// TIA Portal V21 export
FUNCTION "OUTPUT" : Void   // FC4, LAD
{ S7_Optimized_Access := 'TRUE' }
// stored: SetENOAutomatically false
   VAR_TEMP   // added for the SCL form of the ladder/FBD networks
      _w1 : Bool;
   END_VAR
BEGIN

REGION Network 1: VCC PUMP
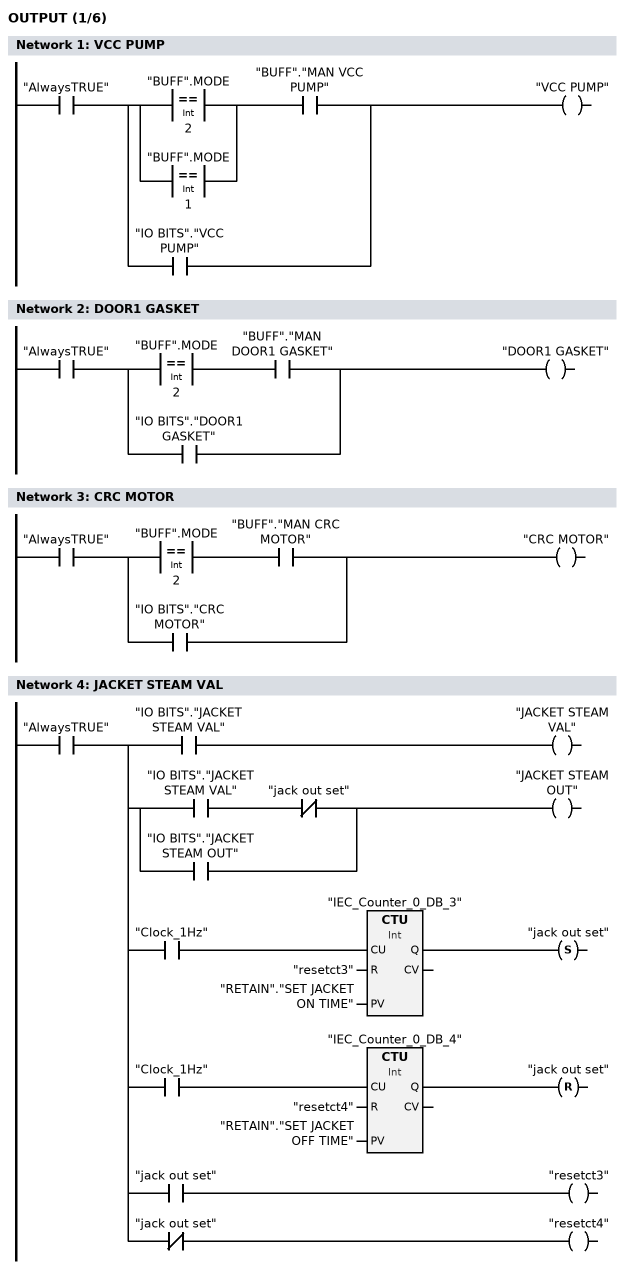
   RUNG wire#powerrail
      Contact( "AlwaysTRUE" )
      wire#w1
      { S7_Templates := "SrcType := Int" } EQ_Contact(in1 := "BUFF".MODE, in2 := 2)
      wire#w2
      Contact( "BUFF"."MAN VCC PUMP" )
      wire#w3
      Coil( "VCC PUMP" )
   END_RUNG
   RUNG wire#w1
      { S7_Templates := "SrcType := Int" } EQ_Contact(in1 := "BUFF".MODE, in2 := 1)
   END_RUNG wire#w2
   RUNG wire#w1
      Contact( "IO BITS"."VCC PUMP" )
   END_RUNG wire#w3
   // the same network as SCL:
   "VCC PUMP" := "AlwaysTRUE" AND (((("BUFF".MODE = 2) OR ("BUFF".MODE = 1)) AND "BUFF"."MAN VCC PUMP") OR "IO BITS"."VCC PUMP");
END_REGION

REGION Network 2: DOOR1 GASKET
   RUNG wire#powerrail
      Contact( "AlwaysTRUE" )
      wire#w1
      { S7_Templates := "SrcType := Int" } EQ_Contact(in1 := "BUFF".MODE, in2 := 2)
      Contact( "BUFF"."MAN DOOR1 GASKET" )
      wire#w2
      Coil( "DOOR1 GASKET" )
   END_RUNG
   RUNG wire#w1
      Contact( "IO BITS"."DOOR1 GASKET" )
   END_RUNG wire#w2
   // the same network as SCL:
   "DOOR1 GASKET" := "AlwaysTRUE" AND ((("BUFF".MODE = 2) AND "BUFF"."MAN DOOR1 GASKET") OR "IO BITS"."DOOR1 GASKET");
END_REGION

REGION Network 3: CRC MOTOR
   RUNG wire#powerrail
      Contact( "AlwaysTRUE" )
      wire#w1
      { S7_Templates := "SrcType := Int" } EQ_Contact(in1 := "BUFF".MODE, in2 := 2)
      Contact( "BUFF"."MAN CRC MOTOR" )
      wire#w2
      Coil( "CRC MOTOR" )
   END_RUNG
   RUNG wire#w1
      Contact( "IO BITS"."CRC MOTOR" )
   END_RUNG wire#w2
   // the same network as SCL:
   "CRC MOTOR" := "AlwaysTRUE" AND ((("BUFF".MODE = 2) AND "BUFF"."MAN CRC MOTOR") OR "IO BITS"."CRC MOTOR");
END_REGION

REGION Network 4: JACKET STEAM VAL
   RUNG wire#powerrail
      Contact( "AlwaysTRUE" )
      wire#w1
      Contact( "IO BITS"."JACKET STEAM VAL" )
      Coil( "JACKET STEAM VAL" )
   END_RUNG
   RUNG wire#w1
      Contact( "IO BITS"."JACKET STEAM VAL" )
      I_Contact( "jack out set" )
      wire#w2
      Coil( "JACKET STEAM OUT" )
   END_RUNG
   RUNG wire#w1
      Contact( "IO BITS"."JACKET STEAM OUT" )
   END_RUNG wire#w2
   RUNG wire#w1
      Contact( "Clock_1Hz" )
      { S7_Templates := "value_type := Int" } "IEC_Counter_0_DB_3".CTU(r := "resetct3", pv := "RETAIN"."SET JACKET ON TIME", cv =>)
      S_Coil( "jack out set" )
   END_RUNG
   RUNG wire#w1
      Contact( "Clock_1Hz" )
      { S7_Templates := "value_type := Int" } "IEC_Counter_0_DB_4".CTU(r := "resetct4", pv := "RETAIN"."SET JACKET OFF TIME", cv =>)
      R_Coil( "jack out set" )
   END_RUNG
   RUNG wire#w1
      Contact( "jack out set" )
      Coil( "resetct3" )
   END_RUNG
   RUNG wire#w1
      I_Contact( "jack out set" )
      Coil( "resetct4" )
   END_RUNG
   // the same network as SCL:
   "JACKET STEAM VAL" := "AlwaysTRUE" AND "IO BITS"."JACKET STEAM VAL";
   "JACKET STEAM OUT" := "AlwaysTRUE" AND (("IO BITS"."JACKET STEAM VAL" AND NOT "jack out set") OR "IO BITS"."JACKET STEAM OUT");
   "IEC_Counter_0_DB_3".CTU(CU := "AlwaysTRUE" AND "Clock_1Hz",
                           R := "resetct3",
                           PV := "RETAIN"."SET JACKET ON TIME");
   IF "IEC_Counter_0_DB_3".Q THEN "jack out set" := TRUE; END_IF;
   "IEC_Counter_0_DB_4".CTU(CU := "AlwaysTRUE" AND "Clock_1Hz",
                           R := "resetct4",
                           PV := "RETAIN"."SET JACKET OFF TIME");
   IF "IEC_Counter_0_DB_4".Q THEN "jack out set" := FALSE; END_IF;
   "resetct3" := "AlwaysTRUE" AND "jack out set";
   "resetct4" := "AlwaysTRUE" AND NOT "jack out set";
END_REGION

REGION Network 5: CHAMBER STEAM VAL
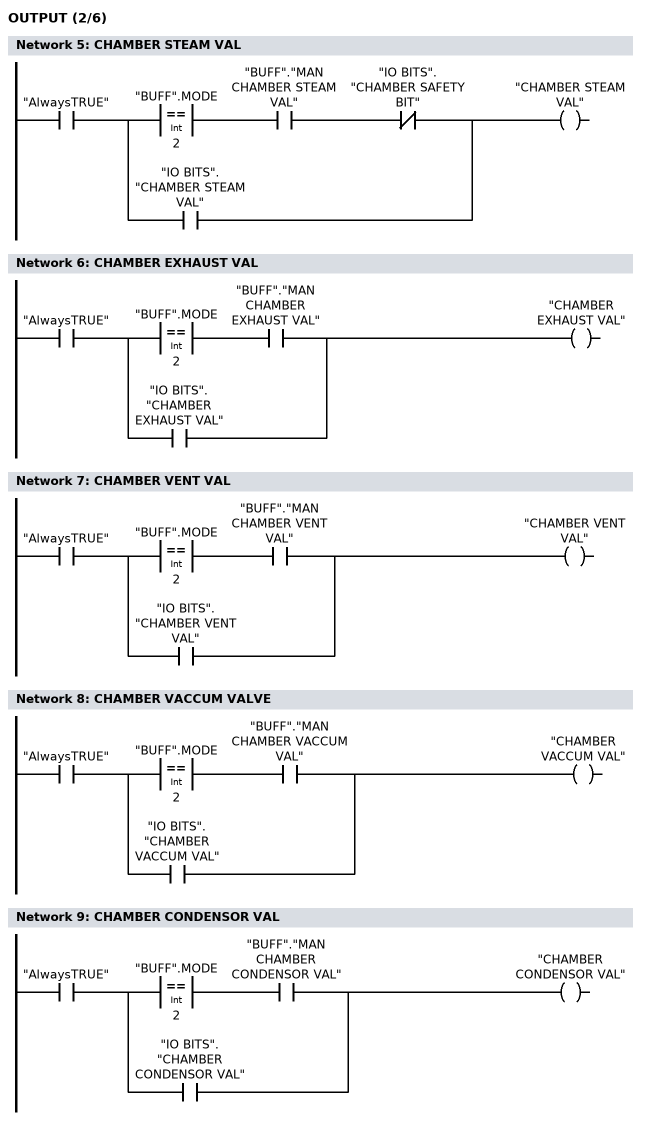
   RUNG wire#powerrail
      Contact( "AlwaysTRUE" )
      wire#w1
      { S7_Templates := "SrcType := Int" } EQ_Contact(in1 := "BUFF".MODE, in2 := 2)
      Contact( "BUFF"."MAN CHAMBER STEAM VAL" )
      I_Contact( "IO BITS"."CHAMBER SAFETY BIT" )
      wire#w2
      Coil( "CHAMBER STEAM VAL" )
   END_RUNG
   RUNG wire#w1
      Contact( "IO BITS"."CHAMBER STEAM VAL" )
   END_RUNG wire#w2
   // the same network as SCL:
   "CHAMBER STEAM VAL" := "AlwaysTRUE" AND ((("BUFF".MODE = 2) AND "BUFF"."MAN CHAMBER STEAM VAL" AND NOT "IO BITS"."CHAMBER SAFETY BIT") OR "IO BITS"."CHAMBER STEAM VAL");
END_REGION

REGION Network 6: CHAMBER EXHAUST VAL
   RUNG wire#powerrail
      Contact( "AlwaysTRUE" )
      wire#w1
      { S7_Templates := "SrcType := Int" } EQ_Contact(in1 := "BUFF".MODE, in2 := 2)
      Contact( "BUFF"."MAN CHAMBER EXHAUST VAL" )
      wire#w2
      Coil( "CHAMBER EXHAUST VAL" )
   END_RUNG
   RUNG wire#w1
      Contact( "IO BITS"."CHAMBER EXHAUST VAL" )
   END_RUNG wire#w2
   // the same network as SCL:
   "CHAMBER EXHAUST VAL" := "AlwaysTRUE" AND ((("BUFF".MODE = 2) AND "BUFF"."MAN CHAMBER EXHAUST VAL") OR "IO BITS"."CHAMBER EXHAUST VAL");
END_REGION

REGION Network 7: CHAMBER VENT VAL
   RUNG wire#powerrail
      Contact( "AlwaysTRUE" )
      wire#w1
      { S7_Templates := "SrcType := Int" } EQ_Contact(in1 := "BUFF".MODE, in2 := 2)
      Contact( "BUFF"."MAN CHAMBER VENT VAL" )
      wire#w2
      Coil( "CHAMBER VENT VAL" )
   END_RUNG
   RUNG wire#w1
      Contact( "IO BITS"."CHAMBER VENT VAL" )
   END_RUNG wire#w2
   // the same network as SCL:
   "CHAMBER VENT VAL" := "AlwaysTRUE" AND ((("BUFF".MODE = 2) AND "BUFF"."MAN CHAMBER VENT VAL") OR "IO BITS"."CHAMBER VENT VAL");
END_REGION

REGION Network 8: CHAMBER VACCUM VALVE
   RUNG wire#powerrail
      Contact( "AlwaysTRUE" )
      wire#w1
      { S7_Templates := "SrcType := Int" } EQ_Contact(in1 := "BUFF".MODE, in2 := 2)
      Contact( "BUFF"."MAN CHAMBER VACCUM VAL" )
      wire#w2
      Coil( "CHAMBER VACCUM VAL" )
   END_RUNG
   RUNG wire#w1
      Contact( "IO BITS"."CHAMBER VACCUM VAL" )
   END_RUNG wire#w2
   // the same network as SCL:
   "CHAMBER VACCUM VAL" := "AlwaysTRUE" AND ((("BUFF".MODE = 2) AND "BUFF"."MAN CHAMBER VACCUM VAL") OR "IO BITS"."CHAMBER VACCUM VAL");
END_REGION

REGION Network 9: CHAMBER CONDENSOR VAL
   RUNG wire#powerrail
      Contact( "AlwaysTRUE" )
      wire#w1
      { S7_Templates := "SrcType := Int" } EQ_Contact(in1 := "BUFF".MODE, in2 := 2)
      Contact( "BUFF"."MAN CHAMBER CONDENSOR VAL" )
      wire#w2
      Coil( "CHAMBER CONDENSOR VAL" )
   END_RUNG
   RUNG wire#w1
      Contact( "IO BITS"."CHAMBER CONDENSOR VAL" )
   END_RUNG wire#w2
   // the same network as SCL:
   "CHAMBER CONDENSOR VAL" := "AlwaysTRUE" AND ((("BUFF".MODE = 2) AND "BUFF"."MAN CHAMBER CONDENSOR VAL") OR "IO BITS"."CHAMBER CONDENSOR VAL");
END_REGION

REGION Network 10: process on lamp
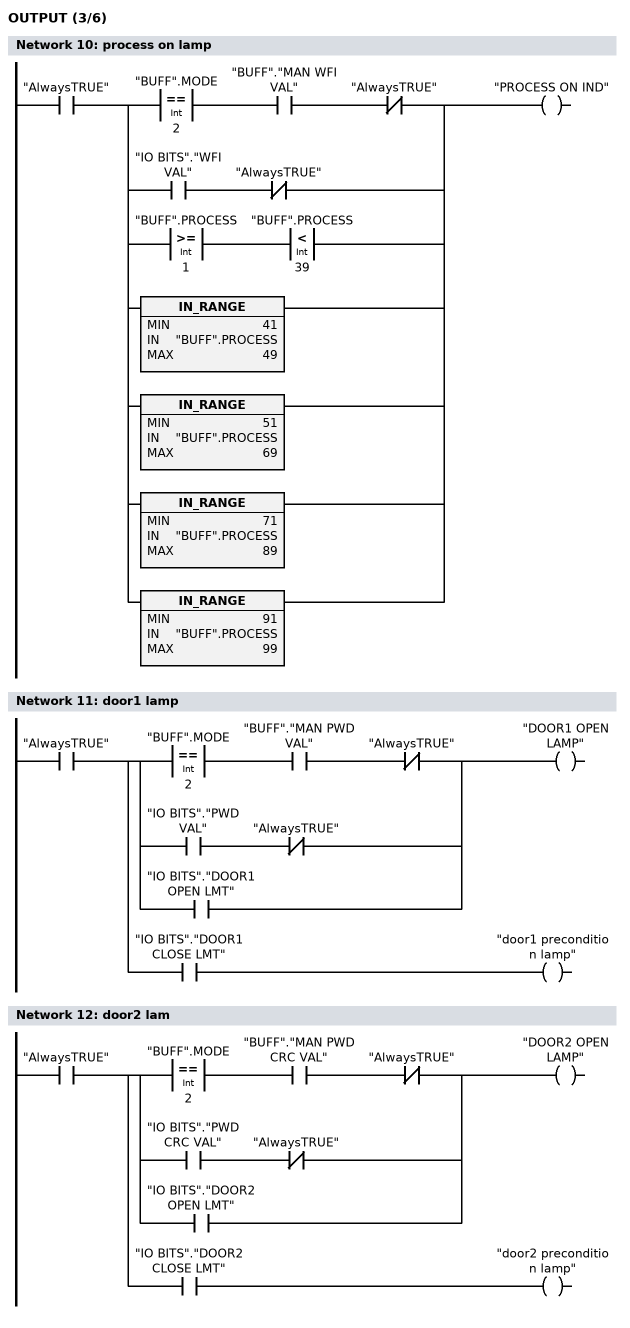
   RUNG wire#powerrail
      Contact( "AlwaysTRUE" )
      wire#w1
      { S7_Templates := "SrcType := Int" } EQ_Contact(in1 := "BUFF".MODE, in2 := 2)
      Contact( "BUFF"."MAN WFI VAL" )
      I_Contact( "AlwaysTRUE" )
      wire#w2
      Coil( "PROCESS ON IND" )
   END_RUNG
   RUNG wire#w1
      Contact( "IO BITS"."WFI VAL" )
      I_Contact( "AlwaysTRUE" )
   END_RUNG wire#w2
   RUNG wire#w1
      { S7_Templates := "SrcType := Int" } GE_Contact(in1 := "BUFF".PROCESS, in2 := 1)
      { S7_Templates := "SrcType := Int" } LT_Contact(in1 := "BUFF".PROCESS, in2 := 39)
   END_RUNG wire#w2
   RUNG wire#w1
      { S7_Templates := "SrcType := Int" } InRange(min := 41, in := "BUFF".PROCESS, max := 49)
   END_RUNG wire#w2
   RUNG wire#w1
      { S7_Templates := "SrcType := Int" } InRange(min := 51, in := "BUFF".PROCESS, max := 69)
   END_RUNG wire#w2
   RUNG wire#w1
      { S7_Templates := "SrcType := Int" } InRange(min := 71, in := "BUFF".PROCESS, max := 89)
   END_RUNG wire#w2
   RUNG wire#w1
      { S7_Templates := "SrcType := Int" } InRange(min := 91, in := "BUFF".PROCESS, max := 99)
   END_RUNG wire#w2
   // the same network as SCL:
   "PROCESS ON IND" := "AlwaysTRUE" AND ((("BUFF".MODE = 2) AND "BUFF"."MAN WFI VAL" AND NOT "AlwaysTRUE") OR ("IO BITS"."WFI VAL" AND NOT "AlwaysTRUE") OR (("BUFF".PROCESS >= 1) AND ("BUFF".PROCESS < 39)) OR ((41 <= "BUFF".PROCESS) AND ("BUFF".PROCESS <= 49)) OR ((51 <= "BUFF".PROCESS) AND ("BUFF".PROCESS <= 69)) OR ((71 <= "BUFF".PROCESS) AND ("BUFF".PROCESS <= 89)) OR ((91 <= "BUFF".PROCESS) AND ("BUFF".PROCESS <= 99)));
END_REGION

REGION Network 11: door1 lamp
   RUNG wire#powerrail
      Contact( "AlwaysTRUE" )
      wire#w1
      { S7_Templates := "SrcType := Int" } EQ_Contact(in1 := "BUFF".MODE, in2 := 2)
      Contact( "BUFF"."MAN PWD VAL" )
      I_Contact( "AlwaysTRUE" )
      wire#w2
      Coil( "DOOR1 OPEN LAMP" )
   END_RUNG
   RUNG wire#w1
      Contact( "IO BITS"."PWD VAL" )
      I_Contact( "AlwaysTRUE" )
   END_RUNG wire#w2
   RUNG wire#w1
      Contact( "IO BITS"."DOOR1 OPEN LMT" )
   END_RUNG wire#w2
   RUNG wire#w1
      Contact( "IO BITS"."DOOR1 CLOSE LMT" )
      Coil( "door1 precondition lamp" )
   END_RUNG
   // the same network as SCL:
   "DOOR1 OPEN LAMP" := "AlwaysTRUE" AND ((("BUFF".MODE = 2) AND "BUFF"."MAN PWD VAL" AND NOT "AlwaysTRUE") OR ("IO BITS"."PWD VAL" AND NOT "AlwaysTRUE") OR "IO BITS"."DOOR1 OPEN LMT");
   "door1 precondition lamp" := "AlwaysTRUE" AND "IO BITS"."DOOR1 CLOSE LMT";
END_REGION

REGION Network 12: door2 lam
   RUNG wire#powerrail
      Contact( "AlwaysTRUE" )
      wire#w1
      { S7_Templates := "SrcType := Int" } EQ_Contact(in1 := "BUFF".MODE, in2 := 2)
      Contact( "BUFF"."MAN PWD CRC VAL" )
      I_Contact( "AlwaysTRUE" )
      wire#w2
      Coil( "DOOR2 OPEN LAMP" )
   END_RUNG
   RUNG wire#w1
      Contact( "IO BITS"."PWD CRC VAL" )
      I_Contact( "AlwaysTRUE" )
   END_RUNG wire#w2
   RUNG wire#w1
      Contact( "IO BITS"."DOOR2 OPEN LMT" )
   END_RUNG wire#w2
   RUNG wire#w1
      Contact( "IO BITS"."DOOR2 CLOSE LMT" )
      Coil( "door2 precondition lamp" )
   END_RUNG
   // the same network as SCL:
   "DOOR2 OPEN LAMP" := "AlwaysTRUE" AND ((("BUFF".MODE = 2) AND "BUFF"."MAN PWD CRC VAL" AND NOT "AlwaysTRUE") OR ("IO BITS"."PWD CRC VAL" AND NOT "AlwaysTRUE") OR "IO BITS"."DOOR2 OPEN LMT");
   "door2 precondition lamp" := "AlwaysTRUE" AND "IO BITS"."DOOR2 CLOSE LMT";
END_REGION

REGION Network 13: DETERGENT DSG VAL
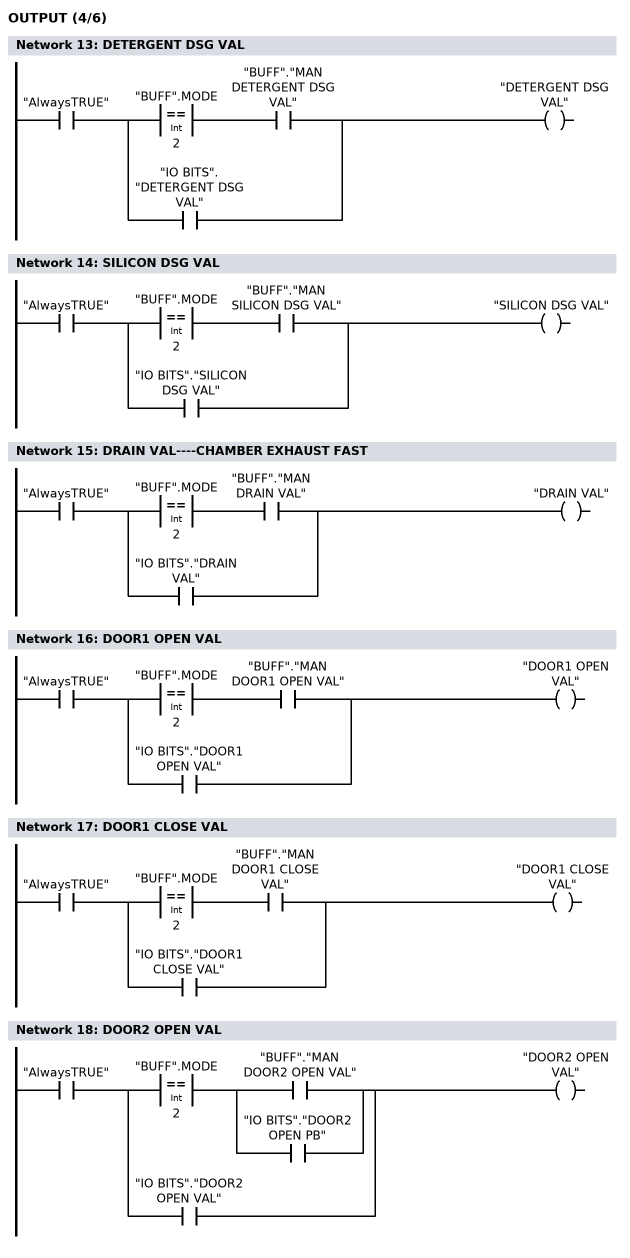
   RUNG wire#powerrail
      Contact( "AlwaysTRUE" )
      wire#w1
      { S7_Templates := "SrcType := Int" } EQ_Contact(in1 := "BUFF".MODE, in2 := 2)
      Contact( "BUFF"."MAN DETERGENT DSG VAL" )
      wire#w2
      Coil( "DETERGENT DSG VAL" )
   END_RUNG
   RUNG wire#w1
      Contact( "IO BITS"."DETERGENT DSG VAL" )
   END_RUNG wire#w2
   // the same network as SCL:
   "DETERGENT DSG VAL" := "AlwaysTRUE" AND ((("BUFF".MODE = 2) AND "BUFF"."MAN DETERGENT DSG VAL") OR "IO BITS"."DETERGENT DSG VAL");
END_REGION

REGION Network 14: SILICON DSG VAL
   RUNG wire#powerrail
      Contact( "AlwaysTRUE" )
      wire#w1
      { S7_Templates := "SrcType := Int" } EQ_Contact(in1 := "BUFF".MODE, in2 := 2)
      Contact( "BUFF"."MAN SILICON DSG VAL" )
      wire#w2
      Coil( "SILICON DSG VAL" )
   END_RUNG
   RUNG wire#w1
      Contact( "IO BITS"."SILICON DSG VAL" )
   END_RUNG wire#w2
   // the same network as SCL:
   "SILICON DSG VAL" := "AlwaysTRUE" AND ((("BUFF".MODE = 2) AND "BUFF"."MAN SILICON DSG VAL") OR "IO BITS"."SILICON DSG VAL");
END_REGION

REGION Network 15: DRAIN VAL----CHAMBER EXHAUST FAST
   RUNG wire#powerrail
      Contact( "AlwaysTRUE" )
      wire#w1
      { S7_Templates := "SrcType := Int" } EQ_Contact(in1 := "BUFF".MODE, in2 := 2)
      Contact( "BUFF"."MAN DRAIN VAL" )
      wire#w2
      Coil( "DRAIN VAL" )
   END_RUNG
   RUNG wire#w1
      Contact( "IO BITS"."DRAIN VAL" )
   END_RUNG wire#w2
   // the same network as SCL:
   "DRAIN VAL" := "AlwaysTRUE" AND ((("BUFF".MODE = 2) AND "BUFF"."MAN DRAIN VAL") OR "IO BITS"."DRAIN VAL");
END_REGION

REGION Network 16: DOOR1 OPEN VAL
   RUNG wire#powerrail
      Contact( "AlwaysTRUE" )
      wire#w1
      { S7_Templates := "SrcType := Int" } EQ_Contact(in1 := "BUFF".MODE, in2 := 2)
      Contact( "BUFF"."MAN DOOR1 OPEN VAL" )
      wire#w2
      Coil( "DOOR1 OPEN VAL" )
   END_RUNG
   RUNG wire#w1
      Contact( "IO BITS"."DOOR1 OPEN VAL" )
   END_RUNG wire#w2
   // the same network as SCL:
   "DOOR1 OPEN VAL" := "AlwaysTRUE" AND ((("BUFF".MODE = 2) AND "BUFF"."MAN DOOR1 OPEN VAL") OR "IO BITS"."DOOR1 OPEN VAL");
END_REGION

REGION Network 17: DOOR1 CLOSE VAL
   RUNG wire#powerrail
      Contact( "AlwaysTRUE" )
      wire#w1
      { S7_Templates := "SrcType := Int" } EQ_Contact(in1 := "BUFF".MODE, in2 := 2)
      Contact( "BUFF"."MAN DOOR1 CLOSE VAL" )
      wire#w2
      Coil( "DOOR1 CLOSE VAL" )
   END_RUNG
   RUNG wire#w1
      Contact( "IO BITS"."DOOR1 CLOSE VAL" )
   END_RUNG wire#w2
   // the same network as SCL:
   "DOOR1 CLOSE VAL" := "AlwaysTRUE" AND ((("BUFF".MODE = 2) AND "BUFF"."MAN DOOR1 CLOSE VAL") OR "IO BITS"."DOOR1 CLOSE VAL");
END_REGION

REGION Network 18: DOOR2 OPEN VAL
   RUNG wire#powerrail
      Contact( "AlwaysTRUE" )
      wire#w1
      { S7_Templates := "SrcType := Int" } EQ_Contact(in1 := "BUFF".MODE, in2 := 2)
      wire#w2
      Contact( "BUFF"."MAN DOOR2 OPEN VAL" )
      wire#w3
      Coil( "DOOR2 OPEN VAL" )
   END_RUNG
   RUNG wire#w2
      Contact( "IO BITS"."DOOR2 OPEN PB" )
   END_RUNG wire#w3
   RUNG wire#w1
      Contact( "IO BITS"."DOOR2 OPEN VAL" )
   END_RUNG wire#w3
   // the same network as SCL:
   "DOOR2 OPEN VAL" := "AlwaysTRUE" AND ((("BUFF".MODE = 2) AND ("BUFF"."MAN DOOR2 OPEN VAL" OR "IO BITS"."DOOR2 OPEN PB")) OR "IO BITS"."DOOR2 OPEN VAL");
END_REGION

REGION Network 19: DOOR2 CLOSE VAL
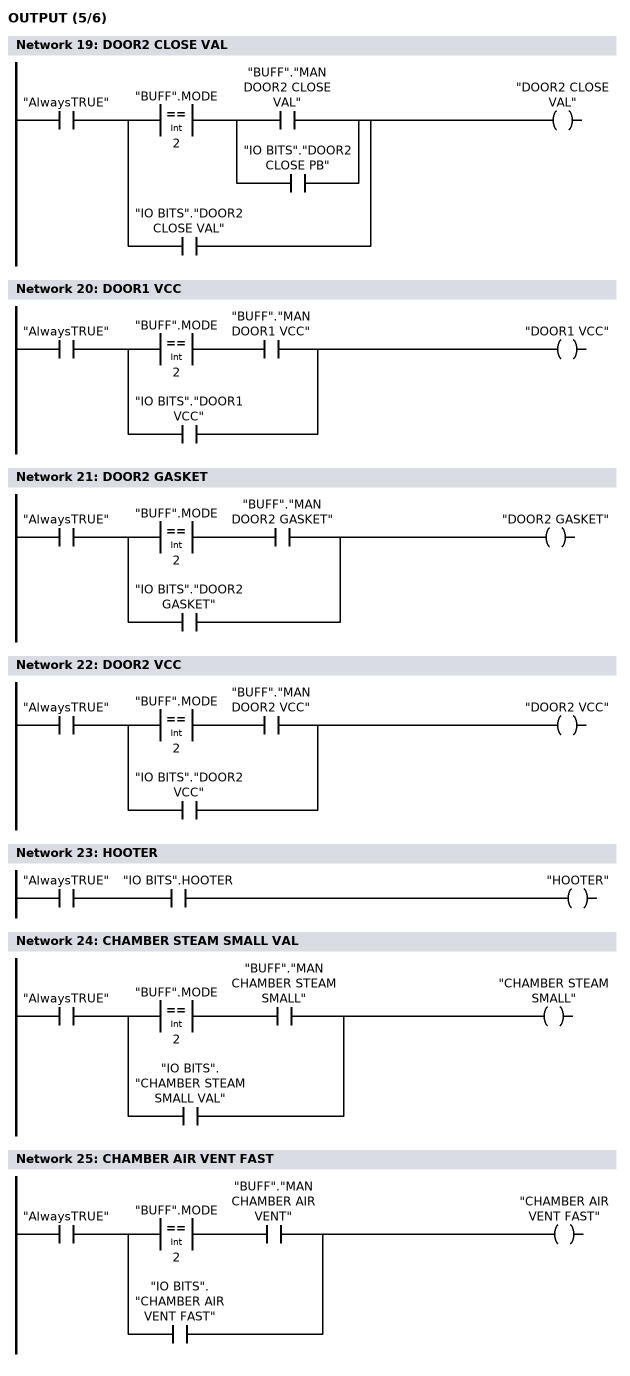
   RUNG wire#powerrail
      Contact( "AlwaysTRUE" )
      wire#w1
      { S7_Templates := "SrcType := Int" } EQ_Contact(in1 := "BUFF".MODE, in2 := 2)
      wire#w2
      Contact( "BUFF"."MAN DOOR2 CLOSE VAL" )
      wire#w3
      Coil( "DOOR2 CLOSE VAL" )
   END_RUNG
   RUNG wire#w2
      Contact( "IO BITS"."DOOR2 CLOSE PB" )
   END_RUNG wire#w3
   RUNG wire#w1
      Contact( "IO BITS"."DOOR2 CLOSE VAL" )
   END_RUNG wire#w3
   // the same network as SCL:
   "DOOR2 CLOSE VAL" := "AlwaysTRUE" AND ((("BUFF".MODE = 2) AND ("BUFF"."MAN DOOR2 CLOSE VAL" OR "IO BITS"."DOOR2 CLOSE PB")) OR "IO BITS"."DOOR2 CLOSE VAL");
END_REGION

REGION Network 20: DOOR1 VCC
   RUNG wire#powerrail
      Contact( "AlwaysTRUE" )
      wire#w1
      { S7_Templates := "SrcType := Int" } EQ_Contact(in1 := "BUFF".MODE, in2 := 2)
      Contact( "BUFF"."MAN DOOR1 VCC" )
      wire#w2
      Coil( "DOOR1 VCC" )
   END_RUNG
   RUNG wire#w1
      Contact( "IO BITS"."DOOR1 VCC" )
   END_RUNG wire#w2
   // the same network as SCL:
   "DOOR1 VCC" := "AlwaysTRUE" AND ((("BUFF".MODE = 2) AND "BUFF"."MAN DOOR1 VCC") OR "IO BITS"."DOOR1 VCC");
END_REGION

REGION Network 21: DOOR2 GASKET
   RUNG wire#powerrail
      Contact( "AlwaysTRUE" )
      wire#w1
      { S7_Templates := "SrcType := Int" } EQ_Contact(in1 := "BUFF".MODE, in2 := 2)
      Contact( "BUFF"."MAN DOOR2 GASKET" )
      wire#w2
      Coil( "DOOR2 GASKET" )
   END_RUNG
   RUNG wire#w1
      Contact( "IO BITS"."DOOR2 GASKET" )
   END_RUNG wire#w2
   // the same network as SCL:
   "DOOR2 GASKET" := "AlwaysTRUE" AND ((("BUFF".MODE = 2) AND "BUFF"."MAN DOOR2 GASKET") OR "IO BITS"."DOOR2 GASKET");
END_REGION

REGION Network 22: DOOR2 VCC
   RUNG wire#powerrail
      Contact( "AlwaysTRUE" )
      wire#w1
      { S7_Templates := "SrcType := Int" } EQ_Contact(in1 := "BUFF".MODE, in2 := 2)
      Contact( "BUFF"."MAN DOOR2 VCC" )
      wire#w2
      Coil( "DOOR2 VCC" )
   END_RUNG
   RUNG wire#w1
      Contact( "IO BITS"."DOOR2 VCC" )
   END_RUNG wire#w2
   // the same network as SCL:
   "DOOR2 VCC" := "AlwaysTRUE" AND ((("BUFF".MODE = 2) AND "BUFF"."MAN DOOR2 VCC") OR "IO BITS"."DOOR2 VCC");
END_REGION

REGION Network 23: HOOTER
   RUNG wire#powerrail
      Contact( "AlwaysTRUE" )
      Contact( "IO BITS".HOOTER )
      Coil( "HOOTER" )
   END_RUNG
   // the same network as SCL:
   "HOOTER" := "AlwaysTRUE" AND "IO BITS".HOOTER;
END_REGION

REGION Network 24: CHAMBER STEAM SMALL VAL
   RUNG wire#powerrail
      Contact( "AlwaysTRUE" )
      wire#w1
      { S7_Templates := "SrcType := Int" } EQ_Contact(in1 := "BUFF".MODE, in2 := 2)
      Contact( "BUFF"."MAN CHAMBER STEAM SMALL" )
      wire#w2
      Coil( "CHAMBER STEAM SMALL" )
   END_RUNG
   RUNG wire#w1
      Contact( "IO BITS"."CHAMBER STEAM SMALL VAL" )
   END_RUNG wire#w2
   // the same network as SCL:
   "CHAMBER STEAM SMALL" := "AlwaysTRUE" AND ((("BUFF".MODE = 2) AND "BUFF"."MAN CHAMBER STEAM SMALL") OR "IO BITS"."CHAMBER STEAM SMALL VAL");
END_REGION

REGION Network 25: CHAMBER AIR VENT FAST
   RUNG wire#powerrail
      Contact( "AlwaysTRUE" )
      wire#w1
      { S7_Templates := "SrcType := Int" } EQ_Contact(in1 := "BUFF".MODE, in2 := 2)
      Contact( "BUFF"."MAN CHAMBER AIR VENT" )
      wire#w2
      Coil( "CHAMBER AIR VENT FAST" )
   END_RUNG
   RUNG wire#w1
      Contact( "IO BITS"."CHAMBER AIR VENT FAST" )
   END_RUNG wire#w2
   // the same network as SCL:
   "CHAMBER AIR VENT FAST" := "AlwaysTRUE" AND ((("BUFF".MODE = 2) AND "BUFF"."MAN CHAMBER AIR VENT") OR "IO BITS"."CHAMBER AIR VENT FAST");
END_REGION

REGION Network 26: BOILER
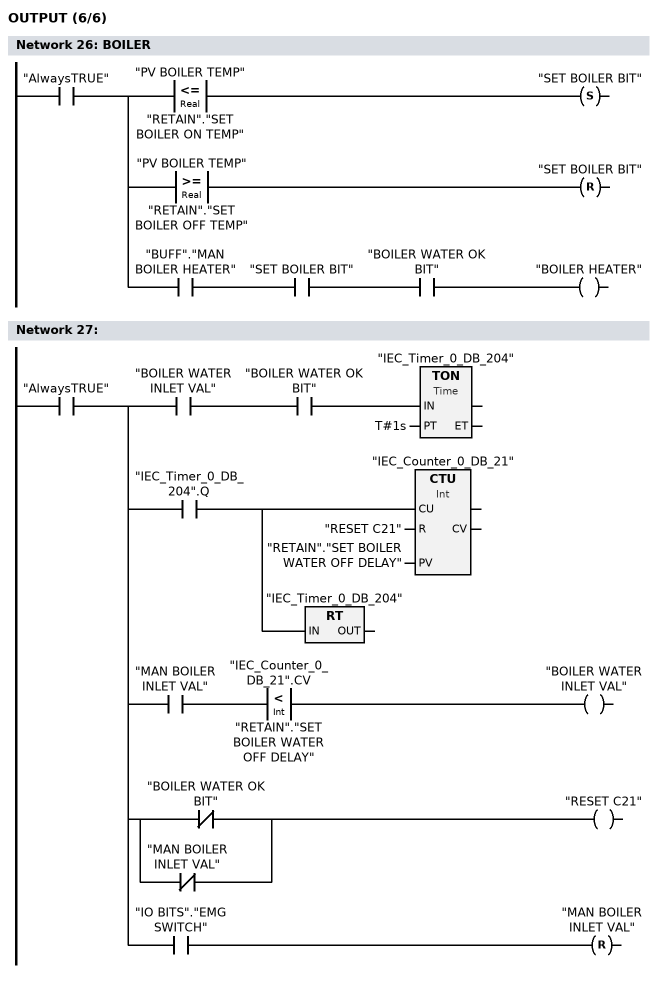
   RUNG wire#powerrail
      Contact( "AlwaysTRUE" )
      wire#w1
      { S7_Templates := "SrcType := Real" } LE_Contact(in1 := "PV BOILER TEMP", in2 := "RETAIN"."SET BOILER ON TEMP")
      S_Coil( "SET BOILER BIT" )
   END_RUNG
   RUNG wire#w1
      { S7_Templates := "SrcType := Real" } GE_Contact(in1 := "PV BOILER TEMP", in2 := "RETAIN"."SET BOILER OFF TEMP")
      R_Coil( "SET BOILER BIT" )
   END_RUNG
   RUNG wire#w1
      Contact( "BUFF"."MAN BOILER HEATER" )
      Contact( "SET BOILER BIT" )
      Contact( "BOILER WATER OK BIT" )
      Coil( "BOILER HEATER" )
   END_RUNG
   // the same network as SCL:
   IF "AlwaysTRUE" AND ("PV BOILER TEMP" <= "RETAIN"."SET BOILER ON TEMP") THEN
       "SET BOILER BIT" := TRUE;
   END_IF;
   IF "AlwaysTRUE" AND ("PV BOILER TEMP" >= "RETAIN"."SET BOILER OFF TEMP") THEN
       "SET BOILER BIT" := FALSE;
   END_IF;
   "BOILER HEATER" := "AlwaysTRUE" AND "BUFF"."MAN BOILER HEATER" AND "SET BOILER BIT" AND "BOILER WATER OK BIT";
END_REGION

REGION Network 27
   RUNG wire#powerrail
      Contact( "AlwaysTRUE" )
      wire#w1
      Contact( "BOILER WATER INLET VAL" )
      Contact( "BOILER WATER OK BIT" )
      { S7_Templates := "time_type := Time" } "IEC_Timer_0_DB_204".TON(pt := T#1s, et =>)
   END_RUNG
   RUNG wire#w1
      Contact( "IEC_Timer_0_DB_204".Q )
      wire#w2
      { S7_Templates := "value_type := Int" } "IEC_Counter_0_DB_21".CTU(r := "RESET C21", pv := "RETAIN"."SET BOILER WATER OFF DELAY", cv =>)
   END_RUNG
   RUNG wire#w2
      RT_Coil( "IEC_Timer_0_DB_204" )
   END_RUNG
   RUNG wire#w1
      Contact( "MAN BOILER INLET VAL" )
      { S7_Templates := "SrcType := Int" } LT_Contact(in1 := "IEC_Counter_0_DB_21".CV, in2 := "RETAIN"."SET BOILER WATER OFF DELAY")
      Coil( "BOILER WATER INLET VAL" )
   END_RUNG
   RUNG wire#w1
      I_Contact( "BOILER WATER OK BIT" )
      wire#w3
      Coil( "RESET C21" )
   END_RUNG
   RUNG wire#w1
      I_Contact( "MAN BOILER INLET VAL" )
   END_RUNG wire#w3
   RUNG wire#w1
      Contact( "IO BITS"."EMG SWITCH" )
      R_Coil( "MAN BOILER INLET VAL" )
   END_RUNG
   // the same network as SCL:
   "IEC_Timer_0_DB_204".TON(IN := "AlwaysTRUE" AND "BOILER WATER INLET VAL" AND "BOILER WATER OK BIT",
                           PT := T#1s);
   #_w1 := "AlwaysTRUE" AND "IEC_Timer_0_DB_204".Q;
   "IEC_Counter_0_DB_21".CTU(CU := #_w1, R := "RESET C21", PV := "RETAIN"."SET BOILER WATER OFF DELAY");
   IF #_w1 THEN RESET_TIMER("IEC_Timer_0_DB_204"); END_IF;
   "BOILER WATER INLET VAL" := "AlwaysTRUE" AND "MAN BOILER INLET VAL" AND ("IEC_Counter_0_DB_21".CV < "RETAIN"."SET BOILER WATER OFF DELAY");
   "RESET C21" := "AlwaysTRUE" AND (NOT "BOILER WATER OK BIT" OR NOT "MAN BOILER INLET VAL");
   IF "AlwaysTRUE" AND "IO BITS"."EMG SWITCH" THEN "MAN BOILER INLET VAL" := FALSE; END_IF;
END_REGION
END_FUNCTION
